# EPICS autosave request: iocBoot/iocUSBTEMP/auto_settings.req
file "USBTEMP_settings.req", P=$(P)
